{attribute 'GeneratedUsingTerminal: EJ1914-0000-0017'}
{attribute addProperty BoxType "EJ1914-0000-0017"}
{attribute addProperty Id "FSOEAT %Q*FSOE_9A7ED3DD7"}
{attribute addProperty CRC "2120688697"}
{attribute addProperty Size "7"}
TYPE FSoE_Outputs_7E672439 :
STRUCT
	{attribute addProperty Name "FSOE"}
	FSOE AT %Q* : FSOE_9A7ED3DD;
END_STRUCT
END_TYPE

(* stored: Version 1.2.0.0, ProductVersion 3.1.4024.9
   DUT FSoE_Outputs_7E672439: Id {746b0258-7efc-466c-9dc0-1b2dd8941c83} *)
